{attribute addProperty BoxType "ELX4181-0000-0016"}
{attribute addProperty Id "AO_OutputsAO_Outputs_F57FA4F9162"}
{attribute addProperty CRC "281800549"}
{attribute addProperty SizeInBites "16"}
{attribute addProperty SizeInBytes "2"}
TYPE Ch_1_10CBEF65 :
STRUCT
	{attribute addProperty Name "AO_Outputs"}
	AO_Outputs  : AO_Outputs_F57FA4F9;
END_STRUCT
END_TYPE

(* stored: Version 1.2.0.0, ProductVersion 3.1.4024.9
   DUT Ch_1_10CBEF65: Id {3f474b59-2c43-44ff-bb27-d78643f395a5} *)
